Staubli VAL3: getFile.pgx

public program getFile(num x_nCamID (dimensions=1), string& x_sActiveJob[] (dimensions=1), bool& x_bError[] (dimensions=1))
begin
  //-----------------------------------------------------------------------
  //Header begin
  //Description of program
  //  Returns the filename of the active job on the In-Sight sensor attached
  //  to camera's ID .
  //
  //  !!!The active job must be saved before this command can be executed
  //  successfully. !!!
  //
  //Input parameters
  //  num x_nCamID :
  //    role : Camera's ID
  //
  //Output parameters
  //  string x_sActiveJob :
  //    role : name of the current active job
  //  bool x_bError :
  //    role : returns true if an error occurred and false otherwise
  //
  //Examples
  //  call getFile(nCamID,l_ActiveJob,x_bError)
  //
  //History
  //  Creation : 19-05-08 - f.Rob
  //Header end
  //-----------------------------------------------------------------------

  nProgram[x_nCamID]=5
  call sendCommand(x_nCamID,"GF",x_bError)
  //No errors
  if !x_bError
    //Read current active job
    call readSocket(x_nCamID,x_sActiveJob,x_bError)
  else
    //Error, no read current active job
    x_sActiveJob=""
  endIf
end
